(* for use with EL3xxx 4-20mA inputs *)
FUNCTION_BLOCK FB_EBUS_420mASensor
VAR_INPUT
	bEnable				: BOOL;		(* TRUE = enable sensor monitoring *)
	bReset				: BOOL;		(* TRUE = reset sensor error *)
	bEnableOverRange	: BOOL;		(* TRUE = enable over-range error *)
	fValueC1			: LREAL;	(* input current 1 (mA) *)
	fValueS1			: LREAL;	(* sensor reading at input voltage 1 *)
	fValueC2			: LREAL;	(* input voltage 2 (mA)  *)
	fValueS2			: LREAL;	(* sensor reading at input voltage 2 *)
	sEtherCATState		: ST_EBUS_EtherCATState;	(* EtherCAT operating state *)
	sDataIn				: ST_EBUS_AnalogueDataIn;	(* input data *)
END_VAR
VAR_OUTPUT
	bStatusOK			: BOOL;		(* comms and sensor status OK *)
	bError				: BOOL;		(* sensor error active *)
	fSensorValue		: LREAL;	(* sensor reading scaled to real units *)
	fmilliAmps			: LREAL;	(* input current *)
END_VAR
VAR
	bCommsStatusOK		: BOOL;
	fbError				: SR;
END_VAR
(*
-------------------------------------------------------------------------------------------------
Date		Version	Author	Comments
-------------------------------------------------------------------------------------------------
30/01/2015	3.00.00	PB		Updated to use ST_EBUS_EtherCATState and ST_EBUS_AnalogueDataIn
							All floating point values now use LREAL

-------------------------------------------------------------------------------------------------
31/03/2010	1.02.00	PB		Initial release

-------------------------------------------------------------------------------------------------
*)

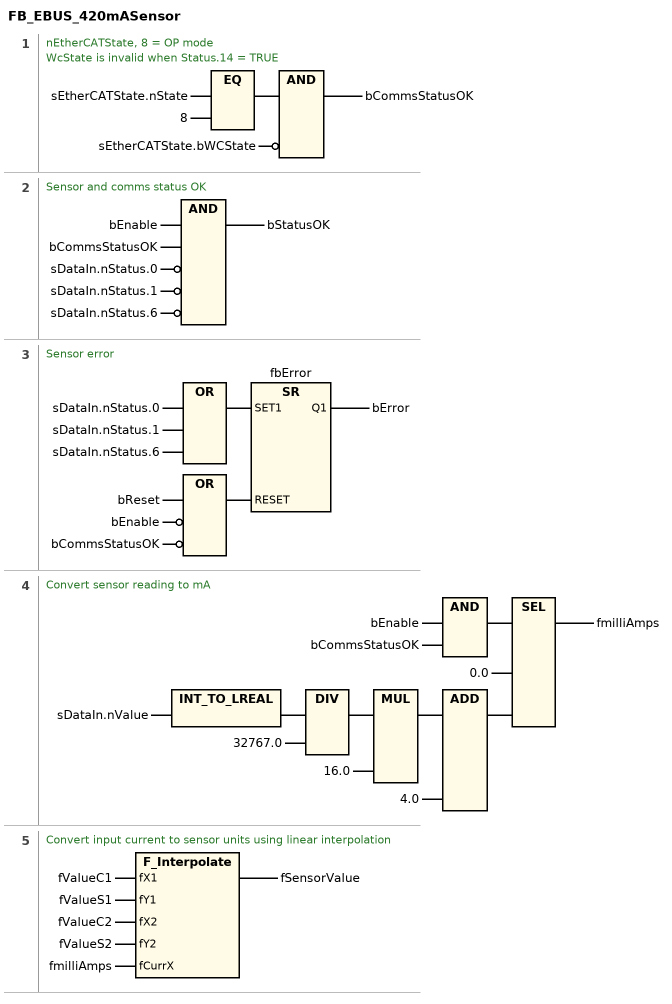
// NETWORK 1
// 					nEtherCATState, 8 = OP mode
// WcState is invalid when Status.14 = TRUE
//
bCommsStatusOK := sEtherCATState.nState = 8 AND NOT sEtherCATState.bWCState;

// NETWORK 2
// Sensor and comms status OK
bStatusOK := bEnable AND bCommsStatusOK AND NOT sDataIn.nStatus.0 AND NOT sDataIn.nStatus.1 AND NOT sDataIn.nStatus.6;

// NETWORK 3
// Sensor error
fbError(SET1 := sDataIn.nStatus.0 OR sDataIn.nStatus.1 OR sDataIn.nStatus.6, RESET := bReset OR NOT bEnable OR NOT bCommsStatusOK); // SR
bError := fbError.Q1;

// NETWORK 4
// Convert sensor reading to mA
fmilliAmps := SEL(bEnable AND bCommsStatusOK, 0.0, (INT_TO_LREAL(sDataIn.nValue) / 32767.0) * 16.0 + 4.0);

// NETWORK 5
// Convert input current to sensor units using linear interpolation
fSensorValue := F_Interpolate(fX1 := fValueC1, fY1 := fValueS1, fX2 := fValueC2, fY2 := fValueS2, fCurrX := fmilliAmps);

END_FUNCTION_BLOCK

(* stored: Version 1.1.0.1, ProductVersion 3.1.4024.15
   POU FB_EBUS_420mASensor: Id {a25748ed-e33c-4b28-b0b5-5080295143e7}, SpecialFunc None *)
